{attribute addProperty BoxType "EPP2816-0008-0018"}
{attribute addProperty Id "DIG_Diag_Inputs_ChannelAT %I*ARRAY[0..8] OF DIG_Diag_Inputs_Channel_AC4A9AF0128160DIG_Inputs_DeviceAT %I*DIG_Inputs_Device_D558E22E4050DIG_Outputs_ChannelAT %Q*ARRAY[0..8] OF DIG_Outputs_Channel_33B76376128160DIG_Outputs_DeviceAT %Q*DIG_Outputs_Device_735003021620WcStateAT %I*WcState_98A4DF7520.250InfoDataAT %I*InfoData_BC63D37F80100"}
{attribute addProperty CRC "1758777227"}
{attribute addProperty SizeInBites "394"}
{attribute addProperty SizeInBytes "49.25"}
TYPE EPP2816_56AF2AEC :
STRUCT
	{attribute addProperty Name "DIG_Diag_Inputs_Channel"}
	DIG_Diag_Inputs_Channel : ARRAY[0..8] OF DIG_Diag_Inputs_Channel_AC4A9AF0;
	{attribute addProperty Name "DIG_Inputs_Device"}
	DIG_Inputs_Device : DIG_Inputs_Device_D558E22E;
	{attribute addProperty Name "DIG_Outputs_Channel"}
	DIG_Outputs_Channel : ARRAY[0..8] OF DIG_Outputs_Channel_33B76376;
	{attribute addProperty Name "DIG_Outputs_Device"}
	DIG_Outputs_Device : DIG_Outputs_Device_73500302;
	{attribute addProperty Name "WcState"}
	WcState : WcState_98A4DF75;
	{attribute addProperty Name "InfoData"}
	InfoData : InfoData_BC63D37F;
END_STRUCT
END_TYPE

(* stored: Version 1.2.0.0, ProductVersion 3.1.4024.9
   DUT EPP2816_56AF2AEC: Id {6cddc2d2-c739-4000-bc12-39be066272bd} *)
